PROGRAM MAIN
VAR
END_VAR

Arbeitsplan();

END_PROGRAM

(* stored: Version 1.1.0.1
   POU MAIN: Id {d55a8836-d109-4370-a4e8-66beca6e2a75}, SpecialFunc None *)
